// TwinCAT 3 PLC project UnitTests
// ProgramVersion: 3.1.4024.0
// libraries:
//   Tc2_Standard, * (Beckhoff Automation GmbH)
//   Tc2_System, * (Beckhoff Automation GmbH)
//   Tc2_Utilities, * (Beckhoff Automation GmbH)
//   Tc3_EventLogger, * (Beckhoff Automation GmbH)
//   Tc3_Module, * (Beckhoff Automation GmbH)
//   tcl_BaseClasses, * (Red Rock Controls Limited)
//   tcl_StringUtils, * (Red Rock Controls Limited)
//   tcl_UnitTestLibrary, * (Red Rock Controls Limited)
// project tree:
//   GVLs/ GlobalNotifications.TcGVL
//   / PlcTask.TcTTO
//   POUs/ MAIN.TcPOU
//   Unit Tests/Execution Result Aggregate/ Test_AggregateResult_Aborted.TcPOU, Test_AggregateResult_Ready.TcPOU, Test_AggregateResult_Busy.TcPOU, Test_AggregateResult_Done.TcPOU, Test_AggregateResult_Error.TcPOU, Test_AggregateResult_ErrorMsg.TcPOU, Test_AggregateResult_Starting.TcPOU, Test_AggregateResult_Aborting.TcPOU
//   Unit Tests/Execution/ Test_TExecutionWhenBusy_Abort_SelectsAborting.TcPOU, Test_TExecutionWhenBusy_SetDone_SetsDone.TcPOU, Test_TExecutionWhenReady_Start_SelectsStarting.TcPOU, Test_TExecution_SetErrorHandlesString_ErrorId.TcPOU
//   Unit Tests/Functions/ Test_ErrorIdToString.TcPOU, Test_F_DINT_TO_UDINT_Conversion.TcPOU, Test_F_Equals.TcPOU, Test_F_NotEqual.TcPOU, Test_F_UDINT_TO_DINT_Conversion.TcPOU
//   Unit Tests/Logger/ Test_TLogger_LogCritical.TcPOU, Test_TLogger_LogError.TcPOU, Test_TLogger_LogWarning.TcPOU, Test_TLogger_LogInfo.TcPOU, Test_TLogger_LogDebug.TcPOU
//   Unit Tests/Notifications/ Test_MultipleNotificationsWithStringArgs.TcPOU, Test_NotificationCountWithQueueingEnabled.TcPOU, Test_NotificationHandlerOnlyAddedOnce.TcPOU, Test_NotificationNoArgs.TcPOU, Test_NotificationWithStringArg.TcPOU
//   Unit Tests/Stream/General/ Test_TStreamBufferResizes.TcPOU
//   Unit Tests/Stream/With alignment checks/ Test_TStreamAddReadArgType_CheckAlignment.TcPOU, Test_TStreamAdd_Read_BLOB_CheckAlignment.TcPOU, Test_TStreamAdd_Read_DINT_CheckAlignment.TcPOU, Test_TStreamAdd_Read_INT_CheckAlignment.TcPOU, Test_TStreamAdd_Read_LINT_CheckAlignment.TcPOU, Test_TStreamAdd_Read_LREAL_CheckAlignment.TcPOU, Test_TStreamAdd_Read_PVOID_CheckAlignment.TcPOU, Test_TStreamAdd_Read_REAL_CheckAlignment.TcPOU, Test_TStreamAdd_Read_UDINT_CheckAlignment.TcPOU, Test_TStreamAdd_Read_UINT_CheckAlignment.TcPOU, Test_TStreamAdd_Read_ULINT_CheckAlignment.TcPOU
//   Unit Tests/Stream/With Arg Type Checking/ Test_TStreamAddReadArgType.TcPOU, Test_TStreamAdd_Read_BLOB.TcPOU, Test_TStreamAdd_Read_BOOL.TcPOU, Test_TStreamAdd_Read_BYTE.TcPOU, Test_TStreamAdd_Read_DINT.TcPOU, Test_TStreamAdd_Read_INT.TcPOU, Test_TStreamAdd_Read_LINT.TcPOU, Test_TStreamAdd_Read_LREAL.TcPOU, Test_TStreamAdd_Read_PVOID.TcPOU, Test_TStreamAdd_Read_REAL.TcPOU, Test_TStreamAdd_Read_Short_STRING.TcPOU, Test_TStreamAdd_Read_STRING.TcPOU, Test_TStreamAdd_Read_T_MaxString.TcPOU, Test_TStreamAdd_Read_UDINT.TcPOU, Test_TStreamAdd_Read_UINT.TcPOU, Test_TStreamAdd_Read_ULINT.TcPOU
//   Unit Tests/ T_TestSuite.TcPOU
// (motion and I/O tree: see PLC project tcl_baseclasses)
// real-time tasks:
//   TASK PlcTask: cycle T#10ms, priority 20, ADS port 350
//   TASK PlcTask1: cycle T#10ms, priority 21, ADS port 351

CONFIGURATION UnitTests
    RESOURCE PLC ON TwinCAT3
        TASK PlcTask(INTERVAL := T#10ms, PRIORITY := 20);
        PROGRAM PB_TestRunner WITH PlcTask : PB_TestRunner;
    END_RESOURCE
END_CONFIGURATION

// ---- GVLs/GlobalNotifications.TcGVL
{attribute 'qualified_only'}
VAR_GLOBAL
	Notification_ExecutionFailed : T_Notification;
	Notification_ExecutionAborted : T_Notification;
	
	
	
	
	
END_VAR

// ---- POUs/MAIN.TcPOU
PROGRAM MAIN
VAR
	TestSuite : T_TestSuite;
END_VAR

TestSuite.RunTests();

END_PROGRAM

// ---- Unit Tests/T_TestSuite.TcPOU
{attribute 'no_explicit_call' := 'do not call this POU directly'}
FUNCTION_BLOCK T_TestSuite
VAR
    Test_AggregateResult_Ready                      : Test_AggregateResult_Ready;
    Test_AggregateResult_Starting                   : Test_AggregateResult_Starting;
    Test_AggregateResult_Busy                       : Test_AggregateResult_Busy;
    Test_AggregateResult_Done                       : Test_AggregateResult_Done;
    Test_AggregateResult_Error                      : Test_AggregateResult_Error;
    Test_AggregateResult_ErrorMsg                   : Test_AggregateResult_ErrorMsg;
    Test_AggregateResult_Aborting                   : Test_AggregateResult_Aborting;
    Test_AggregateResult_Aborted                    : Test_AggregateResult_Aborted;
//    Test_TExecution_WhenBusy_Abort_SelectsAborting  : Test_TExecutionWhenBusy_Abort_SelectsAborting;
//    Test_TExecution_WhenBusy_SetDone_SetsDone       : Test_TExecutionWhenBusy_SetDone_SetsDone;
//    Test_TExecution_WhenReady_Start_SelectsStarting : Test_TExecutionWhenReady_Start_SelectsStarting;
//    Test_TExecution_SetErrorHandlesString_ErrorId   : Test_TExecution_SetErrorHandlesString_ErrorId;
//    Test_F_DINT_TO_UDINT_Conversion                 : Test_F_DINT_TO_UDINT_Conversion;
//    Test_F_UDINT_TO_DINT_Conversion                 : Test_F_UDINT_TO_DINT_Conversion;
//    Test_F_Equals                                   : Test_F_Equals;
//    Test_F_NotEqual                                 : Test_F_NotEqual;
//    Test_ErrorIdToString                            : Test_ErrorIdToString;
//    Test_NotificationNoArgs                         : Test_NotificationNoArgs;
//    Test_NotificationWithStringArg                  : Test_NotificationWithStringArg;
//    Test_NotificationCountWithQueueingEnabled       : Test_NotificationCountWithQueueingEnabled;
//    Test_MultipleNotificationsWithStringArgs        : Test_MultipleNotificationsWithStringArgs;
//    Test_NotificationHandlerOnlyAddedOnce           : Test_NotificationHandlerOnlyAddedOnce;

//    Test_TStreamAdd_Read_BLOB                 : Test_TStreamAdd_Read_BLOB;
//    Test_TStreamAdd_Read_BLOB_CheckAlignment  : Test_TStreamAdd_Read_BLOB_CheckAlignment;
//    Test_TStreamAdd_Read_BOOL                 : Test_TStreamAdd_Read_BOOL;
//    Test_TStreamAdd_Read_BYTE                 : Test_TStreamAdd_Read_BYTE;
//    Test_TStreamAdd_Read_DINT                 : Test_TStreamAdd_Read_DINT;
//    Test_TStreamAdd_Read_DINT_CheckAlignment  : Test_TStreamAdd_Read_DINT_CheckAlignment;
//    Test_TStreamAdd_Read_INT                  : Test_TStreamAdd_Read_INT;
//    Test_TStreamAdd_Read_INT_CheckAlignment   : Test_TStreamAdd_Read_INT_CheckAlignment;
//    Test_TStreamAdd_Read_LINT                 : Test_TStreamAdd_Read_LINT;
//    Test_TStreamAdd_Read_LINT_CheckAlignment  : Test_TStreamAdd_Read_LINT_CheckAlignment;
//    Test_TStreamAdd_Read_LREAL                : Test_TStreamAdd_Read_LREAL;
//    Test_TStreamAdd_Read_LREAL_CheckAlignment : Test_TStreamAdd_Read_LREAL_CheckAlignment;
//    Test_TStreamAdd_Read_PVOID                : Test_TStreamAdd_Read_PVOID;
//    Test_TStreamAdd_Read_PVOID_CheckAlignment : Test_TStreamAdd_Read_PVOID_CheckAlignment;
//    Test_TStreamAdd_Read_REAL                 : Test_TStreamAdd_Read_REAL;
//    Test_TStreamAdd_Read_REAL_CheckAlignment  : Test_TStreamAdd_Read_REAL_CheckAlignment;
//    Test_TStreamAdd_Read_Short_STRING         : Test_TStreamAdd_Read_Short_STRING;
//    Test_TStreamAdd_Read_STRING               : Test_TStreamAdd_Read_STRING;
//    Test_TStreamAdd_Read_T_MaxString          : Test_TStreamAdd_Read_T_MaxString;
//    Test_TStreamAdd_Read_UDINT                : Test_TStreamAdd_Read_UDINT;
//    Test_TStreamAdd_Read_UDINT_CheckAlignment : Test_TStreamAdd_Read_UDINT_CheckAlignment;
//    Test_TStreamAdd_Read_UINT                 : Test_TStreamAdd_Read_UINT;
//    Test_TStreamAdd_Read_UINT_CheckAlignment  : Test_TStreamAdd_Read_UINT_CheckAlignment;
//    Test_TStreamAdd_Read_ULINT                : Test_TStreamAdd_Read_ULINT;
//    Test_TStreamAdd_Read_ULINT_CheckAlignment : Test_TStreamAdd_Read_ULINT_CheckAlignment;
//    Test_TStreamAddReadArgType                : Test_TStreamAddReadArgType;
//    Test_TStreamAddReadArgType_CheckAlignment : Test_TStreamAddReadArgType_CheckAlignment;
//    Test_TStreamBufferResizes                 : Test_TStreamBufferResizes;

//    Test_TLogger_LogCritical : Test_TLogger_LogCritical;
//    Test_TLogger_LogError    : Test_TLogger_LogError;
//    Test_TLogger_LogWarning  : Test_TLogger_LogWarning;
//    Test_TLogger_LogInfo     : Test_TLogger_LogInfo;
//    Test_TLogger_LogDebug    : Test_TLogger_LogDebug;
END_VAR

METHOD RunTests
VAR_INPUT
END_VAR
Test_AggregateResult_Ready                     		.RunTest();
Test_AggregateResult_Starting                       .RunTest();
Test_AggregateResult_Busy                           .RunTest();
Test_AggregateResult_Done                           .RunTest();
Test_AggregateResult_Error                          .RunTest();
Test_AggregateResult_ErrorMsg                       .RunTest();
Test_AggregateResult_Aborting                       .RunTest();
Test_AggregateResult_Aborted                        .RunTest();
//Test_TExecution_WhenBusy_Abort_SelectsAborting      .RunTest();
//Test_TExecution_WhenBusy_SetDone_SetsDone           .RunTest();
//Test_TExecution_WhenReady_Start_SelectsStarting     .RunTest();
//Test_TExecution_SetErrorHandlesString_ErrorId       .RunTest();
//Test_F_DINT_TO_UDINT_Conversion                     .RunTest();
//Test_F_UDINT_TO_DINT_Conversion                     .RunTest();
//Test_F_Equals                                       .RunTest();
//Test_F_NotEqual                                     .RunTest();
//Test_ErrorIdToString                                .RunTest();
//Test_NotificationNoArgs                             .RunTest();
//Test_NotificationWithStringArg                      .RunTest();
//Test_NotificationCountWithQueueingEnabled           .RunTest();
//Test_MultipleNotificationsWithStringArgs            .RunTest();
//Test_NotificationHandlerOnlyAddedOnce               .RunTest();

//Test_TStreamAdd_Read_BLOB                			.RunTest();
//Test_TStreamAdd_Read_BLOB_CheckAlignment            .RunTest();
//Test_TStreamAdd_Read_BOOL                           .RunTest();
//Test_TStreamAdd_Read_BYTE                           .RunTest();
//Test_TStreamAdd_Read_DINT                           .RunTest();
//Test_TStreamAdd_Read_DINT_CheckAlignment            .RunTest();
//Test_TStreamAdd_Read_INT                            .RunTest();
//Test_TStreamAdd_Read_INT_CheckAlignment             .RunTest();
//Test_TStreamAdd_Read_LINT                           .RunTest();
//Test_TStreamAdd_Read_LINT_CheckAlignment            .RunTest();
//Test_TStreamAdd_Read_LREAL                          .RunTest();
//Test_TStreamAdd_Read_LREAL_CheckAlignment           .RunTest();
//Test_TStreamAdd_Read_PVOID                          .RunTest();
//Test_TStreamAdd_Read_PVOID_CheckAlignment           .RunTest();
//Test_TStreamAdd_Read_REAL                           .RunTest();
//Test_TStreamAdd_Read_REAL_CheckAlignment            .RunTest();
//Test_TStreamAdd_Read_Short_STRING                   .RunTest();
//Test_TStreamAdd_Read_STRING                         .RunTest();
//Test_TStreamAdd_Read_T_MaxString                    .RunTest();
//Test_TStreamAdd_Read_UDINT                          .RunTest();
//Test_TStreamAdd_Read_UDINT_CheckAlignment           .RunTest();
//Test_TStreamAdd_Read_UINT                           .RunTest();
//Test_TStreamAdd_Read_UINT_CheckAlignment            .RunTest();
//Test_TStreamAdd_Read_ULINT                          .RunTest();
//Test_TStreamAdd_Read_ULINT_CheckAlignment           .RunTest();
//Test_TStreamAddReadArgType                          .RunTest();
//Test_TStreamAddReadArgType_CheckAlignment           .RunTest();
//Test_TStreamBufferResizes                           .RunTest();

//Test_TLogger_LogCritical .RunTest();
//Test_TLogger_LogError    .RunTest();
//Test_TLogger_LogWarning  .RunTest();
//Test_TLogger_LogInfo     .RunTest();
//Test_TLogger_LogDebug    .RunTest();
END_METHOD

END_FUNCTION_BLOCK

// ---- Unit Tests/Execution Result Aggregate/Test_AggregateResult_Ready.TcPOU
FUNCTION_BLOCK Test_AggregateResult_Ready EXTENDS T_UnitTestBase
VAR
    ResultAggregate : T_ResultAggregate;
    Execution1      : T_Execution;
    Execution2      : T_Execution;
    Execution3      : T_Execution;
END_VAR

{attribute 'analysis' := '-33'} // inhibit unused variable warning
METHOD RunTest
IF Retest THEN
    SUPER^.Init();
END_IF

IF TestCompleted THEN
    RETURN;
END_IF

F_Inc(CycleCount);
IF CycleCount > 1000 THEN
    Fail(Message := 'Timeout');
END_IF

ResultAggregate.Clear();

ResultAggregate.AddResult(Execution1);
ResultAggregate.AddResult(Execution2);
ResultAggregate.AddResult(Execution3);

AssertIsTrue(Condition := ResultAggregate.Ready = TRUE,
             Message   := 'ResultAggregate.Ready is not true');

Execution1.Start();
Execution1.SetBusy();

AssertIsTrue(Condition := ResultAggregate.Ready = FALSE,
             Message   := 'ResultAggregate.Ready is not false');

TestCompleted := TRUE;
END_METHOD

END_FUNCTION_BLOCK

// ---- Unit Tests/Execution Result Aggregate/Test_AggregateResult_Starting.TcPOU
FUNCTION_BLOCK Test_AggregateResult_Starting EXTENDS T_UnitTestBase
VAR
    ResultAggregate : T_ResultAggregate;
    Execution1      : T_Execution;
    Execution2      : T_Execution;
    Execution3      : T_Execution;
END_VAR

{attribute 'analysis' := '-33'} // inhibit unused variable warning
METHOD RunTest
IF Retest THEN
    SUPER^.Init();
END_IF

IF TestCompleted THEN
    RETURN;
END_IF

F_Inc(CycleCount);
IF CycleCount > 1000 THEN
    Fail(Message := 'Timeout');
END_IF

ResultAggregate.Clear();

ResultAggregate.AddResult(Execution1);
ResultAggregate.AddResult(Execution2);
ResultAggregate.AddResult(Execution3);

AssertIsTrue(Condition := ResultAggregate.Starting = FALSE,
             Message   := 'ResultAggregate.Starting is not false');

Execution1.Start();

AssertIsTrue(Condition := ResultAggregate.Starting = TRUE,
             Message   := 'ResultAggregate.Starting is false');

TestCompleted := TRUE;
END_METHOD

END_FUNCTION_BLOCK

// ---- Unit Tests/Execution Result Aggregate/Test_AggregateResult_Busy.TcPOU
FUNCTION_BLOCK Test_AggregateResult_Busy EXTENDS T_UnitTestBase
VAR
	ResultAggregate : T_ResultAggregate;
	Execution1 : T_Execution;
	Execution2 : T_Execution;
	Execution3 : T_Execution;
END_VAR

{attribute 'analysis' := '-33'} // inhibit unused variable warning
METHOD RunTest
IF Retest THEN
    SUPER^.Init();
END_IF

IF TestCompleted THEN
    RETURN;
END_IF

F_Inc(CycleCount);
IF CycleCount > 1000 THEN
    Fail(Message := 'Timeout');
END_IF

ResultAggregate.Clear();

ResultAggregate.AddResult(Execution1);
ResultAggregate.AddResult(Execution2);
ResultAggregate.AddResult(Execution3);

AssertIsTrue(Condition := ResultAggregate.Busy = FALSE,
             Message   := 'ResultAggregate.Busy is not false');

Execution1.Start();
Execution1.SetBusy();

AssertIsTrue(Condition := ResultAggregate.Busy = TRUE,
             Message   := 'ResultAggregate.Busy is false');

TestCompleted := TRUE;
END_METHOD

END_FUNCTION_BLOCK

// ---- Unit Tests/Execution Result Aggregate/Test_AggregateResult_Done.TcPOU
FUNCTION_BLOCK Test_AggregateResult_Done EXTENDS T_UnitTestBase
VAR
	ResultAggregate : T_ResultAggregate;
	Execution1 : T_Execution;
	Execution2 : T_Execution;
	Execution3 : T_Execution;
END_VAR

{attribute 'analysis' := '-33'} // inhibit unused variable warning
METHOD RunTest
IF Retest THEN
    SUPER^.Init();
END_IF

IF TestCompleted THEN
    RETURN;
END_IF

F_Inc(CycleCount);
IF CycleCount > 1000 THEN
    Fail(Message := 'Timeout');
END_IF

ResultAggregate.Clear();

ResultAggregate.AddResult(Execution1);
ResultAggregate.AddResult(Execution2);
ResultAggregate.AddResult(Execution3);

Execution1.Start();
Execution1.SetBusy();
Execution1.SetDone();

Execution2.Start();
Execution2.SetBusy();
Execution2.SetDone();

AssertIsTrue(Condition := ResultAggregate.Done = FALSE,
             Message   := 'ResultAggregate.Done is not false');

Execution3.Start();
Execution3.SetBusy();
Execution3.SetDone();

AssertIsTrue(Condition := ResultAggregate.Done = TRUE,
             Message   := 'ResultAggregate.Done is false');

TestCompleted := TRUE;
END_METHOD

END_FUNCTION_BLOCK

// ---- Unit Tests/Execution Result Aggregate/Test_AggregateResult_Error.TcPOU
FUNCTION_BLOCK Test_AggregateResult_Error EXTENDS T_UnitTestBase
VAR
	ResultAggregate : T_ResultAggregate;
	Execution1 : T_Execution;
	Execution2 : T_Execution;
	Execution3 : T_Execution;
END_VAR

{attribute 'analysis' := '-33'} // inhibit unused variable warning
METHOD RunTest
IF Retest THEN
    SUPER^.Init();
END_IF

IF TestCompleted THEN
    RETURN;
END_IF

F_Inc(CycleCount);
IF CycleCount > 1000 THEN
    Fail(Message := 'Timeout');
END_IF

ResultAggregate.Clear();

ResultAggregate.AddResult(Execution1);
ResultAggregate.AddResult(Execution2);
ResultAggregate.AddResult(Execution3);

Execution1.Start();
Execution1.SetBusy();

AssertIsTrue(Condition := ResultAggregate.Error = FALSE,
             Message   := 'ResultAggregate.Error is not false');

Execution3.Start();
Execution3.SetBusy();
Execution3.SetError('Expected Error Message');

AssertIsTrue(Condition := ResultAggregate.Error = TRUE,
             Message   := 'ResultAggregate.Error is false');

TestCompleted := TRUE;
END_METHOD

END_FUNCTION_BLOCK

// ---- Unit Tests/Execution Result Aggregate/Test_AggregateResult_ErrorMsg.TcPOU
FUNCTION_BLOCK Test_AggregateResult_ErrorMsg EXTENDS T_UnitTestBase
VAR
	ResultAggregate : T_ResultAggregate;
	Execution1 : T_Execution;
	Execution2 : T_Execution;
	Execution3 : T_Execution;
END_VAR

{attribute 'analysis' := '-33'} // inhibit unused variable warning
METHOD RunTest
IF Retest THEN
    SUPER^.Init();
END_IF

IF TestCompleted THEN
    RETURN;
END_IF

F_Inc(CycleCount);
IF CycleCount > 1000 THEN
    Fail(Message := 'Timeout');
END_IF

ResultAggregate.Clear();

ResultAggregate.AddResult(Execution1);
ResultAggregate.AddResult(Execution2);
ResultAggregate.AddResult(Execution3);

Execution1.Start();
Execution1.SetBusy();
Execution1.SetDone();

Execution2.Start();
Execution2.SetBusy();
Execution2.SetDone();

AssertIsTrue(Condition := ResultAggregate.ErrorMsg = '',
             Message   := 'ResultAggregate.ErrorMsg is not blank');

Execution3.Start();
Execution3.SetBusy();
Execution3.SetError('Expected Error Message');

AssertIsTrue(Condition := ResultAggregate.ErrorMsg = 'Expected Error Message',
             Message   := 'ResultAggregate.ErrorMsg is incorrect');

TestCompleted := TRUE;
END_METHOD

END_FUNCTION_BLOCK

// ---- Unit Tests/Execution Result Aggregate/Test_AggregateResult_Aborting.TcPOU
FUNCTION_BLOCK Test_AggregateResult_Aborting EXTENDS T_UnitTestBase
VAR
    ResultAggregate : T_ResultAggregate;
    Execution1      : T_Execution;
    Execution2      : T_Execution;
    Execution3      : T_Execution;
END_VAR

{attribute 'analysis' := '-33'} // inhibit unused variable warning
METHOD RunTest
IF Retest THEN
    SUPER^.Init();
END_IF

IF TestCompleted THEN
    RETURN;
END_IF

F_Inc(CycleCount);
IF CycleCount > 1000 THEN
    Fail(Message := 'Timeout');
END_IF

ResultAggregate.Clear();

ResultAggregate.AddResult(Execution1);
ResultAggregate.AddResult(Execution2);
ResultAggregate.AddResult(Execution3);

AssertIsTrue(Condition := ResultAggregate.Aborting = FALSE,
             Message   := 'ResultAggregate.Aborting is not false');

Execution3.Start();
Execution3.SetBusy();
Execution3.Abort();

AssertIsTrue(Condition := ResultAggregate.Aborting = TRUE,
             Message   := 'ResultAggregate.Aborting is false');

TestCompleted := TRUE;
END_METHOD

END_FUNCTION_BLOCK

// ---- Unit Tests/Execution Result Aggregate/Test_AggregateResult_Aborted.TcPOU
FUNCTION_BLOCK Test_AggregateResult_Aborted EXTENDS T_UnitTestBase
VAR
    ResultAggregate : T_ResultAggregate;
    Execution1      : T_Execution;
    Execution2      : T_Execution;
    Execution3      : T_Execution;
END_VAR

{attribute 'analysis' := '-33'} // inhibit unused variable warning
METHOD RunTest
IF Retest THEN
    SUPER^.Init();
END_IF

IF TestCompleted THEN
    RETURN;
END_IF

F_Inc(CycleCount);
IF CycleCount > 1000 THEN
    Fail(Message := 'Timeout');
END_IF

ResultAggregate.Clear();

ResultAggregate.AddResult(Execution1);
ResultAggregate.AddResult(Execution2);
ResultAggregate.AddResult(Execution3);

AssertIsTrue(Condition := ResultAggregate.Aborted = FALSE,
             Message   := 'ResultAggregate.Aborted is not false');

Execution1.Start();
Execution1.SetBusy();
Execution1.Abort();
Execution1.SetAborted();

Execution2.Start();
Execution2.SetBusy();
Execution2.Abort();
Execution2.SetAborted();

Execution3.Start();
Execution3.SetBusy();
Execution3.Abort();
Execution3.SetAborted();

AssertIsTrue(Condition := ResultAggregate.Aborted,
             Message   := 'ResultAggregate.Aborting is false');

TestCompleted := TRUE;
END_METHOD

END_FUNCTION_BLOCK

// ---- Unit Tests/Execution/Test_TExecutionWhenBusy_Abort_SelectsAborting.TcPOU
FUNCTION_BLOCK Test_TExecutionWhenBusy_Abort_SelectsAborting EXTENDS T_UnitTestbase
VAR
    Execution : T_Execution;
END_VAR

{attribute 'analysis' := '-33'} // inhibit unused variable warning
METHOD RunTest
IF Retest THEN
    SUPER^.Init();
END_IF

IF TestCompleted THEN
    RETURN;
END_IF

F_Inc(CycleCount);
IF CycleCount > 1000 THEN
    Fail(Message := 'Timeout');
END_IF

Execution.Start();
Execution.SetBusy();
Execution.Abort();

AssertIsTrue(Condition := Execution.Aborting,
             Message   := 'Execution.Aborting not true');

TestCompleted := TRUE;
END_METHOD

END_FUNCTION_BLOCK

// ---- Unit Tests/Execution/Test_TExecutionWhenBusy_SetDone_SetsDone.TcPOU
FUNCTION_BLOCK Test_TExecutionWhenBusy_SetDone_SetsDone EXTENDS T_UnitTestbase
VAR
    Execution : T_Execution;
END_VAR

{attribute 'analysis' := '-33'} // inhibit unused variable warning
METHOD RunTest
IF Retest THEN
    SUPER^.Init();
END_IF

IF TestCompleted THEN
    RETURN;
END_IF

F_Inc(CycleCount);
IF CycleCount > 1000 THEN
    Fail(Message := 'Timeout');
END_IF

// Test...
Execution.Start();
Execution.SetBusy();
Execution.SetDone();

AssertIsTrue(Condition := Execution.Done,
             Message   := 'Execution.Done not true');

AssertIsTrue(Condition := Execution.Ready,
             Message   := 'Execution.Ready not true');

TestCompleted := TRUE;
END_METHOD

END_FUNCTION_BLOCK

// ---- Unit Tests/Execution/Test_TExecutionWhenReady_Start_SelectsStarting.TcPOU
FUNCTION_BLOCK Test_TExecutionWhenReady_Start_SelectsStarting EXTENDS T_UnitTestbase
VAR
    Execution : T_Execution;
END_VAR

{attribute 'analysis' := '-33'} // inhibit unused variable warning
METHOD RunTest
IF Retest THEN
    SUPER^.Init();
END_IF

IF TestCompleted THEN
    RETURN;
END_IF

F_Inc(CycleCount);
IF CycleCount > 1000 THEN
    Fail(Message := 'Timeout');
END_IF

// Test...
Execution.Start();

AssertIsTrue(Condition := Execution.Starting,
             Message   := 'Execution.Starting not true');

TestCompleted := TRUE;
END_METHOD

END_FUNCTION_BLOCK

// ---- Unit Tests/Execution/Test_TExecution_SetErrorHandlesString_ErrorId.TcPOU
FUNCTION_BLOCK Test_TExecution_SetErrorHandlesString_ErrorId EXTENDS T_UnitTestBase
VAR
    Execution : T_Execution;
END_VAR
VAR
    ErrorId : STRING := 'Custom error message';
END_VAR

{attribute 'analysis' := '-33'} // inhibit unused variable warning
METHOD RunTest
VAR
    ErrorMsg : STRING := 'Expected error message';
END_VAR
IF Retest THEN
    SUPER^.Init();
END_IF

IF TestCompleted THEN
    RETURN;
END_IF

F_Inc(CycleCount);
IF CycleCount > 1000 THEN
    Fail(Message := 'Timeout');
END_IF

Execution.Start();
Execution.SetBusy();
Execution.SetError(ErrorMsg);

AssertIsTrue(Condition := Execution.ErrorMsg = 'Expected error message',
             Message   := 'Execution.ErrorMsg not correct');

TestCompleted := TRUE;
END_METHOD

END_FUNCTION_BLOCK

// ---- Unit Tests/Functions/Test_ErrorIdToString.TcPOU
FUNCTION_BLOCK Test_ErrorIdToString EXTENDS T_UnitTestBase
VAR_INPUT
END_VAR
VAR_OUTPUT
END_VAR
VAR
END_VAR

{attribute 'analysis' := '-33'} // inhibit unused variable warning
METHOD RunTest
IF Retest THEN
    SUPER^.Init();
END_IF

IF TestCompleted THEN
    RETURN;
END_IF

F_Inc(CycleCount);
IF CycleCount > 1000 THEN
    Fail(Message := 'Timeout');
END_IF

AssertEquals_STRING(Expected := 'Error 0x12BD',
                      Actual   := F_ErrorIdToString(16#12BD),
                      Message  := 'F_ErrorIdToString(16#12BD)');

AssertEquals_STRING(Expected := 'Error 0x12345678',
                      Actual   := F_ErrorIdToString(16#12345678),
                      Message  := 'F_ErrorIdToString(16#12345678)');

AssertEquals_STRING(Expected := 'Error 0x00FF',
                      Actual   := F_ErrorIdToString(16#FF),
                      Message  := 'F_ErrorIdToString(16#FF)');

AssertEquals_STRING(Expected := 'Error 0x0011 - No debugging available',
                      Actual   := F_ErrorIdToString(16#11),
                      Message  := 'F_ErrorIdToString(16#11)');

TestCompleted := TRUE;
END_METHOD

END_FUNCTION_BLOCK

// ---- Unit Tests/Functions/Test_F_DINT_TO_UDINT_Conversion.TcPOU
FUNCTION_BLOCK Test_F_DINT_TO_UDINT_Conversion EXTENDS T_UnitTestBase
VAR
    InputValue     : DINT;
    ConvertedValue : UDINT;
END_VAR

{attribute 'analysis' := '-33'} // inhibit unused variable warning
METHOD RunTest
IF Retest THEN
    SUPER^.Init();
END_IF

IF TestCompleted THEN
    RETURN;
END_IF

F_Inc(CycleCount);
IF CycleCount > 1000 THEN
    Fail(Message := 'Timeout');
END_IF

InputValue     := 2147483648;                  // too big
ConvertedValue := F_UDINT_TO_DINT(InputValue); // limit to largest DINT

AssertEquals_DINT(Expected := 2147483647,
                  Actual   := ConvertedValue,
                  Message  := 'ConvertedValue is not correct');

TestCompleted := TRUE;
END_METHOD

END_FUNCTION_BLOCK

// ---- Unit Tests/Functions/Test_F_Equals.TcPOU
FUNCTION_BLOCK Test_F_Equals EXTENDS T_UnitTestBase
VAR
	
END_VAR

{attribute 'analysis' := '-33'} // inhibit unused variable warning
METHOD RunTest
IF Retest THEN
    SUPER^.Init();
END_IF

IF TestCompleted THEN
    RETURN;
END_IF

F_Inc(CycleCount);
IF CycleCount > 1000 THEN
    Fail(Message := 'Timeout');
END_IF

AssertIsTrue(Condition := F_Equals(1.000_005,
                                   1.000_004,
                                   0.000_002),
             Message := 'F_Equals does not return TRUE');

AssertIsTrue(Condition := NOT F_Equals(1.000_005,
                                   1.000_003,
                                   0.000_001),
             Message := 'F_Equals does not return FALSE');

TestCompleted := TRUE;
END_METHOD

END_FUNCTION_BLOCK

// ---- Unit Tests/Functions/Test_F_NotEqual.TcPOU
FUNCTION_BLOCK Test_F_NotEqual EXTENDS T_UnitTestBase
VAR

END_VAR

{attribute 'analysis' := '-33'} // inhibit unused variable warning
METHOD RunTest
IF Retest THEN
    SUPER^.Init();
END_IF

IF TestCompleted THEN
    RETURN;
END_IF

F_Inc(CycleCount);
IF CycleCount > 1000 THEN
    Fail(Message := 'Timeout');
END_IF

AssertIsTrue(Condition := F_NotEqual(1.000_005,
                                     1.000_003,
                                     0.000_001),
             Message := 'F_NotEquals returns incorrect result');

AssertIsTrue(Condition := NOT F_NotEqual(1.000_005,
                                         1.000_004,
                                         0.000_002),
             Message := 'F_NotEquals returns incorrect result');

TestCompleted := TRUE;
END_METHOD

END_FUNCTION_BLOCK

// ---- Unit Tests/Functions/Test_F_UDINT_TO_DINT_Conversion.TcPOU
FUNCTION_BLOCK Test_F_UDINT_TO_DINT_Conversion EXTENDS T_UnitTestBase
VAR
    InputValue     : UDINT;
    ConvertedValue : DINT;
END_VAR

{attribute 'analysis' := '-33'} // inhibit unused variable warning
METHOD RunTest
IF Retest THEN
    SUPER^.Init();
END_IF

IF TestCompleted THEN
    RETURN;
END_IF

F_Inc(CycleCount);
IF CycleCount > 1000 THEN
    Fail(Message := 'Timeout');
END_IF

InputValue     := UDINT#2147483648;            // too big
ConvertedValue := F_UDINT_TO_DINT(InputValue); // limit to largest DINT

AssertIsTrue(Condition := (ConvertedValue = 2147483647),
             Message   := 'F_UDINT_TO_DINT returns incorrect value');

TestCompleted := TRUE;
END_METHOD

END_FUNCTION_BLOCK

// ---- Unit Tests/Logger/Test_TLogger_LogCritical.TcPOU
FUNCTION_BLOCK Test_TLogger_LogCritical EXTENDS T_UnitTestBase
VAR
    SourceInfo : FB_TcSourceInfo;
END_VAR

{attribute 'analysis' := '-33'} // inhibit unused variable warning
METHOD RunTest
VAR
    ErrorMsg : STRING := 'Expected error message';
END_VAR
IF Retest THEN
    SUPER^.Init();
END_IF

IF TestCompleted THEN
    RETURN;
END_IF

F_Inc(CycleCount);
IF CycleCount > 1000 THEN
    Fail(Message := 'Timeout');
END_IF

SourceInfo.sName := 'ExpectedSourceName';
DefaultLogger.LogCritical(SourceInfo,'Expected critical message1');
DefaultLogger.LogCritical(SourceInfo,'Expected critical message2');

TestCompleted := TRUE;
END_METHOD

END_FUNCTION_BLOCK

// ---- Unit Tests/Logger/Test_TLogger_LogError.TcPOU
FUNCTION_BLOCK Test_TLogger_LogError EXTENDS T_UnitTestBase
VAR
    SourceInfo : FB_TcSourceInfo;
END_VAR

{attribute 'analysis' := '-33'} // inhibit unused variable warning
METHOD RunTest
VAR
    ErrorMsg : STRING := 'Expected error message';
END_VAR
IF Retest THEN
    SUPER^.Init();
END_IF

IF TestCompleted THEN
    RETURN;
END_IF

F_Inc(CycleCount);
IF CycleCount > 1000 THEN
    Fail(Message := 'Timeout');
END_IF

SourceInfo.sName := 'ExpectedSourceName';
DefaultLogger.LogError(SourceInfo,'Expected error message1');
DefaultLogger.LogError(SourceInfo,'Expected error message2');

TestCompleted := TRUE;
END_METHOD

END_FUNCTION_BLOCK

// ---- Unit Tests/Logger/Test_TLogger_LogWarning.TcPOU
FUNCTION_BLOCK Test_TLogger_LogWarning EXTENDS T_UnitTestBase
VAR
    SourceInfo : FB_TcSourceInfo;
END_VAR

{attribute 'analysis' := '-33'} // inhibit unused variable warning
METHOD RunTest
VAR
    ErrorMsg : STRING := 'Expected error message';
END_VAR
IF Retest THEN
    SUPER^.Init();
END_IF

IF TestCompleted THEN
    RETURN;
END_IF

F_Inc(CycleCount);
IF CycleCount > 1000 THEN
    Fail(Message := 'Timeout');
END_IF

SourceInfo.sName := 'ExpectedSourceName';
DefaultLogger.LogWarning(SourceInfo,'Expected warning error message1');
DefaultLogger.LogWarning(SourceInfo,'Expected warning error message2');

TestCompleted := TRUE;
END_METHOD

END_FUNCTION_BLOCK

// ---- Unit Tests/Logger/Test_TLogger_LogInfo.TcPOU
FUNCTION_BLOCK Test_TLogger_LogInfo EXTENDS T_UnitTestBase
VAR
    SourceInfo : FB_TcSourceInfo;
END_VAR

{attribute 'analysis' := '-33'} // inhibit unused variable warning
METHOD RunTest
VAR
    ErrorMsg : STRING := 'Expected error message';
END_VAR
IF Retest THEN
    SUPER^.Init();
END_IF

IF TestCompleted THEN
    RETURN;
END_IF

F_Inc(CycleCount);
IF CycleCount > 1000 THEN
    Fail(Message := 'Timeout');
END_IF

SourceInfo.sName := 'ExpectedSourceName';
DefaultLogger.LogInfo(SourceInfo,'Expected info message1');
DefaultLogger.LogInfo(SourceInfo,'Expected info message2');

TestCompleted := TRUE;
END_METHOD

END_FUNCTION_BLOCK

// ---- Unit Tests/Logger/Test_TLogger_LogDebug.TcPOU
FUNCTION_BLOCK Test_TLogger_LogDebug EXTENDS T_UnitTestBase
VAR
    SourceInfo : FB_TcSourceInfo;
END_VAR

{attribute 'analysis' := '-33'} // inhibit unused variable warning
METHOD RunTest
VAR
    ErrorMsg : STRING := 'Expected error message';
END_VAR
IF Retest THEN
    SUPER^.Init();
END_IF

IF TestCompleted THEN
    RETURN;
END_IF

F_Inc(CycleCount);
IF CycleCount > 1000 THEN
    Fail(Message := 'Timeout');
END_IF

SourceInfo.sName := 'ExpectedSourceName';
DefaultLogger.LogDebug(SourceInfo,'Expected debug message1');
DefaultLogger.LogDebug(SourceInfo,'Expected debug message2');

TestCompleted := TRUE;
END_METHOD

END_FUNCTION_BLOCK

// ---- Unit Tests/Notifications/Test_MultipleNotificationsWithStringArgs.TcPOU
{attribute 'hide'}
FUNCTION_BLOCK Test_MultipleNotificationsWithStringArgs EXTENDS T_UnitTestBase
VAR
    Notification        : T_Notification;
    NotificationHandler : T_NotificationHandler;

    IsRaised          : BOOL;
    NotificationCount : DINT;
END_VAR

{attribute 'analysis' := '-33'} // inhibit unused variable warning
METHOD RunTest
IF Retest THEN
    SUPER^.Init();
END_IF

IF TestCompleted THEN
    RETURN;
END_IF

F_Inc(CycleCount);
IF CycleCount > 1000 THEN
    Fail(Message := 'Timeout');
END_IF

NotificationHandler.NotificationQueueingEnabled := TRUE; // Notification Queuing requires care to ensure all notifications are handled, so disabled by default!

IsRaised          := FALSE;
NotificationCount := 0;

Notification.ClearNotificationHandlers().AddNotificationHandler(NotificationHandler);
Notification.Args.Init(8);

Notification.Args.Clear()
    .Add_INT(1234).Add_STRING('String1');

Notification.Raise();

Notification.Args.Clear()
    .Add_INT(5678).Add_STRING('String2');

Notification.Raise();

AssertEquals_DINT(Expected := 2,
                  Actual   := NotificationHandler.NotificationCount,
                  Message  := 'Handler.NotificationCount is not 2');

AssertIsTrue(Condition := NotificationHandler.IsRaised(),
             Message   := 'NotificationHandler.IsRaised() returns false');

AssertEquals_DINT(Expected := 1,
                  Actual   := NotificationHandler.NotificationCount,
                  Message  := 'Handler.NotificationCount is not 1');

AssertEquals_DINT(Expected := 1234,
                  Actual   := NotificationHandler.Args.Read_INT(),
                  Message  := 'Handler.Args.Read_INT() is not 1234');

AssertEquals_STRING(Expected := 'String1',
                    Actual   := NotificationHandler.Args.Read_STRING(),
                    Message  := 'Handler.Args.Read_STRING() returns incorrect value');

AssertIsTrue(Condition := NotificationHandler.IsRaised(),
             Message   := 'Handler.IsRaised() returns false');

AssertEquals_DINT(Expected := 0,
                  Actual   := NotificationHandler.NotificationCount,
                  Message  := 'Handler.NotificationCount is not 0');

AssertEquals_DINT(Expected := 5678,
                  Actual   := NotificationHandler.Args.Read_INT(),
                  Message  := 'Handler.Args.Read_INT() does not return 5678');

AssertEquals_STRING(Expected := 'String2',
                    Actual   := NotificationHandler.Args.Read_STRING(),
                    Message  := 'Handler.Args.Read_STRING() does not return String2');

AssertIsTrue(Condition := NotificationHandler.IsRaised() = FALSE,
             Message   := 'Handler.IsRaised() return true');

TestCompleted := TRUE;
END_METHOD

END_FUNCTION_BLOCK

// ---- Unit Tests/Notifications/Test_NotificationCountWithQueueingEnabled.TcPOU
FUNCTION_BLOCK Test_NotificationCountWithQueueingEnabled EXTENDS T_UnitTestBase
VAR
    Notification   : T_Notification;
    NotificationHandler : T_NotificationHandler;
    IsRaised : BOOL;
END_VAR

{attribute 'analysis' := '-33'} // inhibit unused variable warning
METHOD RunTest
IF Retest THEN
    SUPER^.Init();
END_IF

IF TestCompleted THEN
    RETURN;
END_IF

F_Inc(CycleCount);
IF CycleCount > 1000 THEN
    Fail(Message := 'Timeout');
END_IF

NotificationHandler.NotificationQueueingEnabled := TRUE; // Notification Queuing requires care to ensure all notifications are handled, so disabled by default!

Notification.ClearNotificationHandlers().AddNotificationHandler(NotificationHandler);

Notification.Raise();
Notification.Raise();
Notification.Raise();

AssertEquals_DINT(Expected := 3,
                  Actual   := NotificationHandler.NotificationCount,
                  Message  := 'Handler.NotificationCount is not 3');

AssertIsTrue(Condition := NotificationHandler.IsRaised(),
             Message   := 'IsRaised() does not return true');

AssertEquals_DINT(Expected := 2,
                  Actual   := NotificationHandler.NotificationCount,
                  Message  := 'Handler.NotificationCount is not 2');

AssertIsTrue(Condition := NotificationHandler.IsRaised(),
             Message   := 'IsRaised() does not return true');

AssertEquals_DINT(Expected := 1,
                  Actual   := NotificationHandler.NotificationCount,
                  Message  := 'Handler.NotificationCount is not 1');

IsRaised := NotificationHandler.IsRaised();

AssertIsTrue(Condition := IsRaised,
             Message   := 'IsRaised is false');

AssertEquals_DINT(Expected     := 0,
                  Actual       := NotificationHandler.NotificationCount,
                  Message := 'Handler.NotificationCount is not 0');

AssertIsTrue(Condition    := NotificationHandler.IsRaised() = FALSE,
             Message := 'Handler.IsRaised() is not false');

TestCompleted := TRUE;
END_METHOD

END_FUNCTION_BLOCK

// ---- Unit Tests/Notifications/Test_NotificationHandlerOnlyAddedOnce.TcPOU
FUNCTION_BLOCK Test_NotificationHandlerOnlyAddedOnce EXTENDS T_UnitTestBase
VAR
    Notification        : T_Notification;
    NotificationHandler : T_NotificationHandler;
    IsRaised            : BOOL;
END_VAR

{attribute 'analysis' := '-33'} // inhibit unused variable warning
METHOD RunTest
IF Retest THEN
    SUPER^.Init();
END_IF

IF TestCompleted THEN
    RETURN;
END_IF

F_Inc(CycleCount);
IF CycleCount > 1000 THEN
    Fail(Message := 'Timeout');
END_IF

Notification
    .ClearNotificationHandlers()
    .AddNotificationHandler(NotificationHandler)
    .AddNotificationHandler(NotificationHandler);

Notification.Raise();
IsRaised := NotificationHandler.IsRaised();

AssertIsTrue(Condition := IsRaised = TRUE,
             Message   := 'IsRaised is not true');

IsRaised := NotificationHandler.IsRaised();

AssertIsTrue(Condition := IsRaised = FALSE,
             Message   := 'IsRaised is not false');

TestCompleted := TRUE;
END_METHOD

END_FUNCTION_BLOCK

// ---- Unit Tests/Notifications/Test_NotificationNoArgs.TcPOU
FUNCTION_BLOCK Test_NotificationNoArgs EXTENDS T_UnitTestBase
VAR
    Notification        : T_Notification;
    NotificationHandler : T_NotificationHandler;
    IsRaised            : BOOL;
END_VAR

{attribute 'analysis' := '-33'} // inhibit unused variable warning
METHOD RunTest
IF Retest THEN
    SUPER^.Init();
END_IF

IF TestCompleted THEN
    RETURN;
END_IF

F_Inc(CycleCount);
IF CycleCount > 1000 THEN
    Fail(Message := 'Timeout');
END_IF

Notification.ClearNotificationHandlers().AddNotificationHandler(NotificationHandler);

Notification.Raise();
IsRaised := NotificationHandler.IsRaised();

AssertIsTrue(Condition := IsRaised,
             Message   := 'IsRaised is not true');

TestCompleted := TRUE;
END_METHOD

END_FUNCTION_BLOCK

// ---- Unit Tests/Notifications/Test_NotificationWithStringArg.TcPOU
{attribute 'hide'}
FUNCTION_BLOCK Test_NotificationWithStringArg EXTENDS T_UnitTestBase
VAR
    Notification        : T_Notification;
    NotificationHandler : T_NotificationHandler;

    ResultString : T_MaxString;
    Args         : I_StreamReader;
    IsRaised     : BOOL;
END_VAR

{attribute 'analysis' := '-33'} // inhibit unused variable warning
METHOD RunTest
IF Retest THEN
    SUPER^.Init();
END_IF

IF TestCompleted THEN
    RETURN;
END_IF

F_Inc(CycleCount);
IF CycleCount > 1000 THEN
    Fail(Message := 'Timeout');
END_IF

Notification.ClearNotificationHandlers().AddNotificationHandler(NotificationHandler);
Notification.Args.Init(81);

Notification.Args.Clear().Add_STRING('Big long string passed to the notification handler for later use');
Notification.Raise();

IF NotificationHandler.IsRaised() THEN
    Args         := NotificationHandler.Args;
    ResultString := Args.Read_STRING();
END_IF

AssertEquals_STRING(Expected := 'Big long string passed to the notification handler for later use',
                    Actual   := ResultString,
                    Message  := 'ResultString is not correct');

TestCompleted := TRUE;
END_METHOD

END_FUNCTION_BLOCK

// ---- Unit Tests/Stream/General/Test_TStreamBufferResizes.TcPOU
FUNCTION_BLOCK Test_TStreamBufferResizes EXTENDS T_UnitTestBase
VAR
    Stream : T_Stream(StreamLength := 2);
END_VAR

{attribute 'analysis' := '-33'} // inhibit unused variable warning
METHOD RunTest
IF Retest THEN
    SUPER^.Init();
END_IF

IF TestCompleted THEN
    RETURN;
END_IF

F_Inc(CycleCount);
IF CycleCount > 1000 THEN
    Fail(Message := 'Timeout');
END_IF

Stream.Init(2);

Stream.Add_INT(1234);
Stream.Add_INT(1235);
Stream.Add_INT(1236);
Stream.Add_INT(1237);

AssertEquals_UDINT(Expected     := 8,
                   Actual       := Stream.WritePosition,
                   Message := 'Stream.WritePosition');

AssertEquals_UDINT(Expected     := 8,
                   Actual       := Stream.StreamLength,
                   Message := 'Stream.StreamLength');

Stream.SetReadPosition(0);

AssertEquals_INT(Expected     := 1234,
                 Actual       := Stream.Read_INT(),
                 Message := 'Stream.ReadInt()');

AssertEquals_UDINT(Expected     := 2,
                   Actual       := Stream.ReadPosition,
                   Message := 'Stream.ReadPosition');

TestCompleted := TRUE;
END_METHOD

END_FUNCTION_BLOCK

// ---- Unit Tests/Stream/With alignment checks/Test_TStreamAddReadArgType_CheckAlignment.TcPOU
FUNCTION_BLOCK Test_TStreamAddReadArgType_CheckAlignment EXTENDS T_UnitTestBase
VAR
    Stream : T_Stream(StreamLength := 2);
END_VAR

{attribute 'analysis' := '-33'} // inhibit unused variable warning
METHOD RunTest
IF Retest THEN
    SUPER^.Init();
END_IF

IF TestCompleted THEN
    RETURN;
END_IF

F_Inc(CycleCount);
IF CycleCount > 1000 THEN
    Fail(Message := 'Timeout');
END_IF

Stream.Init(2);

Stream.Add_BYTE(123); // add a byte to test alignment checks...
Stream.SetNextArgTypeId(E_ArgTypeId.Type_LINT);

AssertEquals_UDINT(Expected := 4,
                   Actual   := Stream.WritePosition,
                   Message  := 'Stream.WritePosition');

Stream.SetReadPosition(0);

Stream.Read_BYTE();

AssertEquals_INT(Expected := E_ArgTypeId.Type_LINT,
                 Actual   := Stream.GetNextArgTypeId(),
                 Message  := 'Stream.GetNextArgTypeId()');

AssertEquals_UDINT(Expected := 4,
                   Actual   := Stream.ReadPosition,
                   Message  := 'Stream.ReadPosition');

TestCompleted := TRUE;
END_METHOD

END_FUNCTION_BLOCK

// ---- Unit Tests/Stream/With alignment checks/Test_TStreamAdd_Read_BLOB_CheckAlignment.TcPOU
FUNCTION_BLOCK Test_TStreamAdd_Read_BLOB_CheckAlignment EXTENDS T_UnitTestBase
VAR
    Stream : T_Stream(StreamLength := 2);
    Now    : TIMESTRUCT := (wDay := 23,
        wMonth := 12,
        wYear := 1945,
        wHour := 22,
        wMinute := 20,
        wSecond := 18);
    NowFromStream : TIMESTRUCT;

    LREAL_Value : LREAL := 1.234;
END_VAR

{attribute 'analysis' := '-33'} // inhibit unused variable warning
METHOD RunTest
IF Retest THEN
    SUPER^.Init();
END_IF

IF TestCompleted THEN
    RETURN;
END_IF

F_Inc(CycleCount);
IF CycleCount > 1000 THEN
    Fail(Message := 'Timeout');
END_IF

Stream.Init(2);
NowFromStream.wDay    := 0;
NowFromStream.wMonth  := 0;
NowFromStream.wYear   := 0;
NowFromStream.wHour   := 0;
NowFromStream.wMinute := 0;
NowFromStream.wSecond := 0;

Stream.Add_BYTE(123);// add a byte to test alignment checks...
Stream.Add_BLOB(Now);

Stream.SetReadPosition(0);
Stream.Read_BYTE();
Stream.Read_BLOB(NowFromStream);

// check the value...
AssertEquals_ANY(Expected     := Now,
                            Actual       := NowFromStream,
                            Message := 'NowFromStream');

// check we are at the end of the stream..							
AssertEquals_UDINT(Expected     := Stream.StreamLength,
                             Actual       := Stream.ReadPosition,
                             Message := 'Stream.ReadPosition');

TestCompleted := TRUE;
END_METHOD

END_FUNCTION_BLOCK

// ---- Unit Tests/Stream/With alignment checks/Test_TStreamAdd_Read_DINT_CheckAlignment.TcPOU
FUNCTION_BLOCK Test_TStreamAdd_Read_DINT_CheckAlignment EXTENDS T_UnitTestBase
VAR
    Stream  : T_Stream(StreamLength := 2);
    ArgType : E_ArgTypeId := E_ArgTypeId.Type_DINT;
END_VAR

{attribute 'analysis' := '-33'} // inhibit unused variable warning
METHOD RunTest
IF Retest THEN
    SUPER^.Init();
END_IF

IF TestCompleted THEN
    RETURN;
END_IF

F_Inc(CycleCount);
IF CycleCount > 1000 THEN
    Fail(Message := 'Timeout');
END_IF

Stream.Init(2);

Stream.Add_BYTE(123);// add a byte to test alignment checks...
Stream.Add_DINT(12345678);

Stream.SetReadPosition(0);

Stream.Read_BYTE();

// check next value...	
AssertEquals_DINT(Expected     := 12345678,
                            Actual       := Stream.Read_DINT(),
                            Message := 'Stream.Read_DINT()');

// check we are at the end of the stream..							
AssertEquals_UDINT(Expected     := Stream.StreamLength,
                             Actual       := Stream.ReadPosition,
                             Message := 'Stream.ReadPosition');

TestCompleted := TRUE;
END_METHOD

END_FUNCTION_BLOCK

// ---- Unit Tests/Stream/With alignment checks/Test_TStreamAdd_Read_INT_CheckAlignment.TcPOU
FUNCTION_BLOCK Test_TStreamAdd_Read_INT_CheckAlignment EXTENDS T_UnitTestBase
VAR
    Stream  : T_Stream(StreamLength := 2);
    ArgType : E_ArgTypeId := E_ArgTypeId.Type_INT;
END_VAR

{attribute 'analysis' := '-33'} // inhibit unused variable warning
METHOD RunTest
IF Retest THEN
    SUPER^.Init();
END_IF

IF TestCompleted THEN
    RETURN;
END_IF

F_Inc(CycleCount);
IF CycleCount > 1000 THEN
    Fail(Message := 'Timeout');
END_IF

Stream.Init(2);

Stream.Add_BYTE(123);// add a byte to test alignment checks...
Stream.Add_INT(1234);

Stream.SetReadPosition(0);

Stream.Read_BYTE();

// check next value...	
AssertEquals_INT(Expected     := 1234,
                           Actual       := Stream.Read_INT(),
                           Message := 'Stream.Read_INT()');

// check we are at the end of the stream..							
AssertEquals_UDINT(Expected     := Stream.StreamLength,
                             Actual       := Stream.ReadPosition,
                             Message := 'Stream.ReadPosition');

TestCompleted := TRUE;
END_METHOD

END_FUNCTION_BLOCK

// ---- Unit Tests/Stream/With alignment checks/Test_TStreamAdd_Read_LINT_CheckAlignment.TcPOU
FUNCTION_BLOCK Test_TStreamAdd_Read_LINT_CheckAlignment EXTENDS T_UnitTestBase
VAR
    Stream  : T_Stream(StreamLength := 2);
    ArgType : E_ArgTypeId := E_ArgTypeId.Type_LINT;
END_VAR

{attribute 'analysis' := '-33'} // inhibit unused variable warning
METHOD RunTest
IF Retest THEN
    SUPER^.Init();
END_IF

IF TestCompleted THEN
    RETURN;
END_IF

F_Inc(CycleCount);
IF CycleCount > 1000 THEN
    Fail(Message := 'Timeout');
END_IF

Stream.Init(2);

Stream.Add_BYTE(123);// add a byte to test alignment checks...
Stream.Add_LINT(123456789);

Stream.SetReadPosition(0);

Stream.Read_BYTE();

// check next value...	
AssertEquals_LINT(Expected     := 123456789,
                            Actual       := Stream.Read_LINT(),
                            Message := 'Stream.Read_LINT()');

// check we are at the end of the stream..							
AssertEquals_UDINT(Expected     := Stream.StreamLength,
                             Actual       := Stream.ReadPosition,
                             Message := 'Stream.ReadPosition');

TestCompleted := TRUE;
END_METHOD

END_FUNCTION_BLOCK

// ---- Unit Tests/Stream/With alignment checks/Test_TStreamAdd_Read_LREAL_CheckAlignment.TcPOU
FUNCTION_BLOCK Test_TStreamAdd_Read_LREAL_CheckAlignment EXTENDS T_UnitTestBase
VAR
    Stream  : T_Stream(StreamLength := 2);
    ArgType : E_ArgTypeId := E_ArgTypeId.Type_LREAL;
END_VAR

{attribute 'analysis' := '-33'} // inhibit unused variable warning
METHOD RunTest
IF Retest THEN
    SUPER^.Init();
END_IF

IF TestCompleted THEN
    RETURN;
END_IF

F_Inc(CycleCount);
IF CycleCount > 1000 THEN
    Fail(Message := 'Timeout');
END_IF

Stream.Init(2);

Stream.Add_BYTE(123);// add a byte to test alignment checks...
Stream.Add_LREAL(1.234567891234);

Stream.SetReadPosition(0);

Stream.Read_BYTE();

// check next value...	
AssertEquals_LREAL(Expected     := 1.234567891234,
                             Actual       := Stream.Read_LREAL(),
                             Delta        := 0.000000000001,
                             Message := 'Stream.Read_LREAL()');

// check we are at the end of the stream..							
AssertEquals_UDINT(Expected     := Stream.StreamLength,
                             Actual       := Stream.ReadPosition,
                             Message := 'Stream.ReadPosition');

TestCompleted := TRUE;
END_METHOD

END_FUNCTION_BLOCK

// ---- Unit Tests/Stream/With alignment checks/Test_TStreamAdd_Read_PVOID_CheckAlignment.TcPOU
FUNCTION_BLOCK Test_TStreamAdd_Read_PVOID_CheckAlignment EXTENDS T_UnitTestBase
VAR
    Stream  : T_Stream(StreamLength := 2);
    ArgType : E_ArgTypeId := E_ArgTypeId.Type_PVOID;
    Bob     : INT;
END_VAR

{attribute 'analysis' := '-33'} // inhibit unused variable warning
METHOD RunTest
IF Retest THEN
    SUPER^.Init();
END_IF

IF TestCompleted THEN
    RETURN;
END_IF

F_Inc(CycleCount);
IF CycleCount > 1000 THEN
    Fail(Message := 'Timeout');
END_IF

Stream.Init(2);

Stream.Add_BYTE(123);// add a byte to test alignment checks...
Stream.Add_PVOID(ADR(Bob));

Stream.SetReadPosition(0);

Stream.Read_BYTE();

// check next value...	
AssertEquals_PVOID(Expected     := ADR(Bob),
                             Actual       := Stream.Read_PVOID(),
                             Message := 'Stream.Read_PVOID()');

// check we are at the end of the stream..							
AssertEquals_UDINT(Expected     := Stream.StreamLength,
                             Actual       := Stream.ReadPosition,
                             Message := 'Stream.ReadPosition');

TestCompleted := TRUE;
END_METHOD

END_FUNCTION_BLOCK

// ---- Unit Tests/Stream/With alignment checks/Test_TStreamAdd_Read_REAL_CheckAlignment.TcPOU
FUNCTION_BLOCK Test_TStreamAdd_Read_REAL_CheckAlignment EXTENDS T_UnitTestBase
VAR
    Stream  : T_Stream(StreamLength := 2);
    ArgType : E_ArgTypeId := E_ArgTypeId.Type_REAL;
END_VAR

{attribute 'analysis' := '-33'} // inhibit unused variable warning
METHOD RunTest
IF Retest THEN
    SUPER^.Init();
END_IF

IF TestCompleted THEN
    RETURN;
END_IF

F_Inc(CycleCount);
IF CycleCount > 1000 THEN
    Fail(Message := 'Timeout');
END_IF

Stream.Init(2);

Stream.Add_BYTE(123);// add a byte to test alignment checks...
Stream.Add_REAL(1.234567);

Stream.SetReadPosition(0);

Stream.Read_BYTE();

// check next value...	
AssertEquals_REAL(Expected     := 1.234567,
                            Actual       := Stream.Read_REAL(),
                            Delta        := 0.000001,
                            Message := 'Stream.Read_REAL()');

// check we are at the end of the stream..							
AssertEquals_UDINT(Expected     := Stream.StreamLength,
                             Actual       := Stream.ReadPosition,
                             Message := 'Stream.ReadPosition');

TestCompleted := TRUE;
END_METHOD

END_FUNCTION_BLOCK

// ---- Unit Tests/Stream/With alignment checks/Test_TStreamAdd_Read_UDINT_CheckAlignment.TcPOU
FUNCTION_BLOCK Test_TStreamAdd_Read_UDINT_CheckAlignment EXTENDS T_UnitTestBase
VAR
    Stream  : T_Stream(StreamLength := 2);
    ArgType : E_ArgTypeId := E_ArgTypeId.Type_UDINT;
END_VAR

{attribute 'analysis' := '-33'} // inhibit unused variable warning
METHOD RunTest
IF Retest THEN
    SUPER^.Init();
END_IF

IF TestCompleted THEN
    RETURN;
END_IF

F_Inc(CycleCount);
IF CycleCount > 1000 THEN
    Fail(Message := 'Timeout');
END_IF

Stream.Init(2);

Stream.Add_BYTE(123);// add a byte to test alignment checks...
Stream.Add_UDINT(12345678);

Stream.SetReadPosition(0);

Stream.Read_BYTE();

// check next value...	
AssertEquals_UDINT(Expected     := 12345678,
                             Actual       := Stream.Read_UDINT(),
                             Message := 'Stream.Read_UDINT()');

// check we are at the end of the stream..							
AssertEquals_UDINT(Expected     := Stream.StreamLength,
                             Actual       := Stream.ReadPosition,
                             Message := 'Stream.ReadPosition');

TestCompleted := TRUE;
END_METHOD

END_FUNCTION_BLOCK

// ---- Unit Tests/Stream/With alignment checks/Test_TStreamAdd_Read_UINT_CheckAlignment.TcPOU
FUNCTION_BLOCK Test_TStreamAdd_Read_UINT_CheckAlignment EXTENDS T_UnitTestBase
VAR
    Stream  : T_Stream(StreamLength := 2);
    ArgType : E_ArgTypeId := E_ArgTypeId.Type_UINT;
END_VAR

{attribute 'analysis' := '-33'} // inhibit unused variable warning
METHOD RunTest
IF Retest THEN
    SUPER^.Init();
END_IF

IF TestCompleted THEN
    RETURN;
END_IF

F_Inc(CycleCount);
IF CycleCount > 1000 THEN
    Fail(Message := 'Timeout');
END_IF

Stream.Init(2);

Stream.Add_BYTE(123);// add a byte to test alignment checks...
Stream.Add_UINT(4567);

Stream.SetReadPosition(0);

Stream.Read_BYTE();

// check next value...	
AssertEquals_UINT(Expected     := 4567,
                            Actual       := Stream.Read_UINT(),
                            Message := 'Stream.Read_UINT()');

// check we are at the end of the stream..							
AssertEquals_UDINT(Expected     := Stream.StreamLength,
                             Actual       := Stream.ReadPosition,
                             Message := 'Stream.ReadPosition');

TestCompleted := TRUE;
END_METHOD

END_FUNCTION_BLOCK

// ---- Unit Tests/Stream/With alignment checks/Test_TStreamAdd_Read_ULINT_CheckAlignment.TcPOU
FUNCTION_BLOCK Test_TStreamAdd_Read_ULINT_CheckAlignment EXTENDS T_UnitTestBase
VAR
    Stream  : T_Stream(StreamLength := 2);
    ArgType : E_ArgTypeId := E_ArgTypeId.Type_ULINT;
END_VAR

{attribute 'analysis' := '-33'} // inhibit unused variable warning
METHOD RunTest
IF Retest THEN
    SUPER^.Init();
END_IF

IF TestCompleted THEN
    RETURN;
END_IF

F_Inc(CycleCount);
IF CycleCount > 1000 THEN
    Fail(Message := 'Timeout');
END_IF


Stream.Init(2);

Stream.Add_BYTE(123); // add a byte to test alignment checks...
Stream.Add_ULINT(123456789);

Stream.SetReadPosition(0);

Stream.Read_BYTE();

// check next value...	
AssertEquals_ULINT(Expected     := 123456789,
                   Actual       := Stream.Read_ULINT(),
                   Message := 'Stream.Read_ULINT()');

// check we are at the end of the stream..							
AssertEquals_UDINT(Expected     := Stream.StreamLength,
                   Actual       := Stream.ReadPosition,
                   Message := 'Stream.ReadPosition');

TestCompleted := TRUE;
END_METHOD

END_FUNCTION_BLOCK

// ---- Unit Tests/Stream/With Arg Type Checking/Test_TStreamAddReadArgType.TcPOU
FUNCTION_BLOCK Test_TStreamAddReadArgType EXTENDS T_UnitTestBase
VAR
    Stream : T_Stream(StreamLength := 2);
END_VAR

{attribute 'analysis' := '-33'} // inhibit unused variable warning
METHOD RunTest
IF Retest THEN
    SUPER^.Init();
END_IF

IF TestCompleted THEN
    RETURN;
END_IF

F_Inc(CycleCount);
IF CycleCount > 1000 THEN
    Fail(Message := 'Timeout');
END_IF

Stream.Init(2);

Stream.SetNextArgTypeId(E_ArgTypeId.Type_LINT);

AssertEquals_UDINT(Expected     := 2,
                             Actual       := Stream.WritePosition,
                             Message := 'Stream.WritePosition');

Stream.SetReadPosition(0);

AssertEquals_INT(Expected     := E_ArgTypeId.Type_LINT,
                           Actual       := Stream.GetNextArgTypeId(),
                           Message := 'Stream.GetNextArgTypeId()');

AssertEquals_UDINT(Expected     := 2,
                             Actual       := Stream.ReadPosition,
                             Message := 'Stream.ReadPosition');

TestCompleted := TRUE;
END_METHOD

END_FUNCTION_BLOCK

// ---- Unit Tests/Stream/With Arg Type Checking/Test_TStreamAdd_Read_BLOB.TcPOU
FUNCTION_BLOCK Test_TStreamAdd_Read_BLOB EXTENDS T_UnitTestBase
VAR
    Stream : T_Stream(StreamLength := 2);
    Now    : TIMESTRUCT := (wDay := 23,
        wMonth := 12,
        wYear := 1945,
        wHour := 22,
        wMinute := 20,
        wSecond := 18);
    NowFromStream : TIMESTRUCT;

    LREAL_Value : LREAL := 1.234;
END_VAR

{attribute 'analysis' := '-33'} // inhibit unused variable warning
METHOD RunTest
IF Retest THEN
    SUPER^.Init();
END_IF

IF TestCompleted THEN
    RETURN;
END_IF

F_Inc(CycleCount);
IF CycleCount > 1000 THEN
    Fail(Message := 'Timeout');
END_IF

Stream.Init(2);
NowFromStream.wDay    := 0;
NowFromStream.wMonth  := 0;
NowFromStream.wYear   := 0;
NowFromStream.wHour   := 0;
NowFromStream.wMinute := 0;
NowFromStream.wSecond := 0;

Stream.SetNextArgTypeId(E_ArgTypeId.Type_Blob);
Stream.Add_BLOB(Now);

Stream.SetReadPosition(0);

IF Stream.GetNextArgTypeId() = E_ArgTypeId.Type_Blob THEN
    Stream.Read_BLOB(NowFromStream);
END_IF

// check the value...
AssertEquals_ANY(Expected     := Now,
                            Actual       := NowFromStream,
                            Message := 'NowFromStream');

// check we are at the end of the stream..							
AssertEquals_UDINT(Expected     := Stream.StreamLength,
                             Actual       := Stream.ReadPosition,
                             Message := 'Stream.ReadPosition');

TestCompleted := TRUE;
END_METHOD

END_FUNCTION_BLOCK

// ---- Unit Tests/Stream/With Arg Type Checking/Test_TStreamAdd_Read_BOOL.TcPOU
FUNCTION_BLOCK Test_TStreamAdd_Read_BOOL EXTENDS T_UnitTestBase
VAR
    Stream  : T_Stream(StreamLength := 2);
    ArgType : E_ArgTypeId := E_ArgTypeId.Type_BOOL;
END_VAR

{attribute 'analysis' := '-33'} // inhibit unused variable warning
METHOD RunTest
IF Retest THEN
    SUPER^.Init();
END_IF

IF TestCompleted THEN
    RETURN;
END_IF

F_Inc(CycleCount);
IF CycleCount > 1000 THEN
    Fail(Message := 'Timeout');
END_IF

Stream.Init(2);

// add a bool...
Stream.SetNextArgTypeId(ArgType);
Stream.Add_BOOL(TRUE);

Stream.SetReadPosition(0);

// check next arg type is correct...
AssertEquals_INT(Expected     := ArgType,
                           Actual       := Stream.GetNextArgTypeId(),
                           Message := 'Stream.GetNextArgTypeId()');

// check next value...	
AssertEquals_BOOL(Expected     := TRUE,
                            Actual       := Stream.Read_BOOL(),
                            Message := 'Stream.Read_BOOL()');

// check we are at the end of the stream..							
AssertEquals_UDINT(Expected     := Stream.StreamLength,
                             Actual       := Stream.ReadPosition,
                             Message := 'Stream.ReadPosition');

TestCompleted := TRUE;
END_METHOD

END_FUNCTION_BLOCK

// ---- Unit Tests/Stream/With Arg Type Checking/Test_TStreamAdd_Read_BYTE.TcPOU
FUNCTION_BLOCK Test_TStreamAdd_Read_BYTE EXTENDS T_UnitTestBase
VAR
    Stream  : T_Stream(StreamLength := 2);
    ArgType : E_ArgTypeId := E_ArgTypeId.Type_BYTE;
END_VAR

{attribute 'analysis' := '-33'} // inhibit unused variable warning
METHOD RunTest
IF Retest THEN
    SUPER^.Init();
END_IF

IF TestCompleted THEN
    RETURN;
END_IF

F_Inc(CycleCount);
IF CycleCount > 1000 THEN
    Fail(Message := 'Timeout');
END_IF

Stream.Init(2);

// add a byte...
Stream.SetNextArgTypeId(ArgType);
Stream.Add_BYTE(123);

Stream.SetReadPosition(0);

// check next arg type is correct...
AssertEquals_INT(Expected     := ArgType,
                           Actual       := Stream.GetNextArgTypeId(),
                           Message := 'Stream.GetNextArgTypeId()');

// check next value...	
AssertEquals_BYTE(Expected     := 123,
                            Actual       := Stream.Read_BYTE(),
                            Message := 'Stream.Read_BYTE()');

// check we are at the end of the stream..							
AssertEquals_UDINT(Expected     := Stream.StreamLength,
                             Actual       := Stream.ReadPosition,
                             Message := 'Stream.ReadPosition');

TestCompleted := TRUE;
END_METHOD

END_FUNCTION_BLOCK

// ---- Unit Tests/Stream/With Arg Type Checking/Test_TStreamAdd_Read_DINT.TcPOU
FUNCTION_BLOCK Test_TStreamAdd_Read_DINT EXTENDS T_UnitTestBase
VAR
    Stream  : T_Stream(StreamLength := 2);
    ArgType : E_ArgTypeId := E_ArgTypeId.Type_DINT;
END_VAR

{attribute 'analysis' := '-33'} // inhibit unused variable warning
METHOD RunTest
IF Retest THEN
    SUPER^.Init();
END_IF

IF TestCompleted THEN
    RETURN;
END_IF

F_Inc(CycleCount);
IF CycleCount > 1000 THEN
    Fail(Message := 'Timeout');
END_IF

Stream.Init(2);

// add a DINT...
Stream.SetNextArgTypeId(ArgType);
Stream.Add_DINT(12345678);

Stream.SetReadPosition(0);

// check next arg type is correct...
AssertEquals_INT(Expected     := ArgType,
                           Actual       := Stream.GetNextArgTypeId(),
                           Message := 'Stream.GetNextArgTypeId()');

// check next value...	
AssertEquals_DINT(Expected     := 12345678,
                            Actual       := Stream.Read_DINT(),
                            Message := 'Stream.Read_DINT()');

// check we are at the end of the stream..							
AssertEquals_UDINT(Expected     := Stream.StreamLength,
                             Actual       := Stream.ReadPosition,
                             Message := 'Stream.ReadPosition');

TestCompleted := TRUE;
END_METHOD

END_FUNCTION_BLOCK

// ---- Unit Tests/Stream/With Arg Type Checking/Test_TStreamAdd_Read_INT.TcPOU
FUNCTION_BLOCK Test_TStreamAdd_Read_INT EXTENDS T_UnitTestBase
VAR
    Stream  : T_Stream(StreamLength := 2);
    ArgType : E_ArgTypeId := E_ArgTypeId.Type_INT;
END_VAR

{attribute 'analysis' := '-33'} // inhibit unused variable warning
METHOD RunTest
IF Retest THEN
    SUPER^.Init();
END_IF

IF TestCompleted THEN
    RETURN;
END_IF

F_Inc(CycleCount);
IF CycleCount > 1000 THEN
    Fail(Message := 'Timeout');
END_IF

Stream.Init(2);

// add an INT...
Stream.SetNextArgTypeId(ArgType);
Stream.Add_INT(1234);

Stream.SetReadPosition(0);

// check next arg type is correct...
AssertEquals_INT(Expected     := ArgType,
                           Actual       := Stream.GetNextArgTypeId(),
                           Message := 'Stream.GetNextArgTypeId()');

// check next value...	
AssertEquals_INT(Expected     := 1234,
                           Actual       := Stream.Read_INT(),
                           Message := 'Stream.Read_INT()');

// check we are at the end of the stream..							
AssertEquals_UDINT(Expected     := Stream.StreamLength,
                             Actual       := Stream.ReadPosition,
                             Message := 'Stream.ReadPosition');

TestCompleted := TRUE;
END_METHOD

END_FUNCTION_BLOCK

// ---- Unit Tests/Stream/With Arg Type Checking/Test_TStreamAdd_Read_LINT.TcPOU
FUNCTION_BLOCK Test_TStreamAdd_Read_LINT EXTENDS T_UnitTestBase
VAR
    Stream  : T_Stream(StreamLength := 2);
    ArgType : E_ArgTypeId := E_ArgTypeId.Type_LINT;
END_VAR

{attribute 'analysis' := '-33'} // inhibit unused variable warning
METHOD RunTest
IF Retest THEN
    SUPER^.Init();
END_IF

IF TestCompleted THEN
    RETURN;
END_IF

F_Inc(CycleCount);
IF CycleCount > 1000 THEN
    Fail(Message := 'Timeout');
END_IF

Stream.Init(2);

// add a LINT...
Stream.SetNextArgTypeId(ArgType);
Stream.Add_LINT(123456789);

Stream.SetReadPosition(0);

// check next arg type is correct...
AssertEquals_INT(Expected     := ArgType,
                           Actual       := Stream.GetNextArgTypeId(),
                           Message := 'Stream.GetNextArgTypeId()');

// check next value...	
AssertEquals_LINT(Expected     := 123456789,
                            Actual       := Stream.Read_LINT(),
                            Message := 'Stream.Read_LINT()');

// check we are at the end of the stream..							
AssertEquals_UDINT(Expected     := Stream.StreamLength,
                             Actual       := Stream.ReadPosition,
                             Message := 'Stream.ReadPosition');

TestCompleted := TRUE;
END_METHOD

END_FUNCTION_BLOCK

// ---- Unit Tests/Stream/With Arg Type Checking/Test_TStreamAdd_Read_LREAL.TcPOU
FUNCTION_BLOCK Test_TStreamAdd_Read_LREAL EXTENDS T_UnitTestBase
VAR
    Stream  : T_Stream(StreamLength := 2);
    ArgType : E_ArgTypeId := E_ArgTypeId.Type_LREAL;
END_VAR

{attribute 'analysis' := '-33'} // inhibit unused variable warning
METHOD RunTest
IF Retest THEN
    SUPER^.Init();
END_IF

IF TestCompleted THEN
    RETURN;
END_IF

F_Inc(CycleCount);
IF CycleCount > 1000 THEN
    Fail(Message := 'Timeout');
END_IF

Stream.Init(2);

// add a LREAL...
Stream.SetNextArgTypeId(ArgType);
Stream.Add_LREAL(1.234567891234);

Stream.SetReadPosition(0);

// check next arg type is correct...
AssertEquals_INT(Expected     := ArgType,
                           Actual       := Stream.GetNextArgTypeId(),
                           Message := 'Stream.GetNextArgTypeId()');

// check next value...	
AssertEquals_LREAL(Expected     := 1.234567891234,
                             Actual       := Stream.Read_LREAL(),
                             Delta        := 0.000000000001,
                             Message := 'Stream.Read_LREAL()');

// check we are at the end of the stream..							
AssertEquals_UDINT(Expected     := Stream.StreamLength,
                             Actual       := Stream.ReadPosition,
                             Message := 'Stream.ReadPosition');

TestCompleted := TRUE;
END_METHOD

END_FUNCTION_BLOCK

// ---- Unit Tests/Stream/With Arg Type Checking/Test_TStreamAdd_Read_PVOID.TcPOU
FUNCTION_BLOCK Test_TStreamAdd_Read_PVOID EXTENDS T_UnitTestBase
VAR
    Stream  : T_Stream(StreamLength := 2);
    ArgType : E_ArgTypeId := E_ArgTypeId.Type_PVOID;
    Bob     : INT;
END_VAR

{attribute 'analysis' := '-33'} // inhibit unused variable warning
METHOD RunTest
IF Retest THEN
    SUPER^.Init();
END_IF

IF TestCompleted THEN
    RETURN;
END_IF

F_Inc(CycleCount);
IF CycleCount > 1000 THEN
    Fail(Message := 'Timeout');
END_IF

Stream.Init(2);

// add a pointer...
Stream.SetNextArgTypeId(ArgType);
Stream.Add_PVOID(ADR(Bob));

Stream.SetReadPosition(0);

// check next arg type is correct...
AssertEquals_INT(Expected     := ArgType,
                           Actual       := Stream.GetNextArgTypeId(),
                           Message := 'Stream.GetNextArgTypeId()');

// check next value...	
AssertEquals_PVOID(Expected     := ADR(Bob),
                             Actual       := Stream.Read_PVOID(),
                             Message := 'Stream.Read_PVOID()');

// check we are at the end of the stream..							
AssertEquals_UDINT(Expected     := Stream.StreamLength,
                             Actual       := Stream.ReadPosition,
                             Message := 'Stream.ReadPosition');

TestCompleted := TRUE;
END_METHOD

END_FUNCTION_BLOCK

// ---- Unit Tests/Stream/With Arg Type Checking/Test_TStreamAdd_Read_REAL.TcPOU
FUNCTION_BLOCK Test_TStreamAdd_Read_REAL EXTENDS T_UnitTestBase
VAR
    Stream  : T_Stream(StreamLength := 2);
    ArgType : E_ArgTypeId := E_ArgTypeId.Type_REAL;
END_VAR

{attribute 'analysis' := '-33'} // inhibit unused variable warning
METHOD RunTest
IF Retest THEN
    SUPER^.Init();
END_IF

IF TestCompleted THEN
    RETURN;
END_IF

F_Inc(CycleCount);
IF CycleCount > 1000 THEN
    Fail(Message := 'Timeout');
END_IF

Stream.Init(2);

// add a REAL...
Stream.SetNextArgTypeId(ArgType);
Stream.Add_REAL(1.234567);

Stream.SetReadPosition(0);

// check next arg type is correct...
AssertEquals_INT(Expected     := ArgType,
                           Actual       := Stream.GetNextArgTypeId(),
                           Message := 'Stream.GetNextArgTypeId()');

// check next value...	
AssertEquals_REAL(Expected     := 1.234567,
                            Actual       := Stream.Read_REAL(),
                            Delta        := 0.000001,
                            Message := 'Stream.Read_REAL()');

// check we are at the end of the stream..							
AssertEquals_UDINT(Expected     := Stream.StreamLength,
                             Actual       := Stream.ReadPosition,
                             Message := 'Stream.ReadPosition');

TestCompleted := TRUE;
END_METHOD

END_FUNCTION_BLOCK

// ---- Unit Tests/Stream/With Arg Type Checking/Test_TStreamAdd_Read_Short_STRING.TcPOU
FUNCTION_BLOCK Test_TStreamAdd_Read_Short_STRING EXTENDS T_UnitTestBase
VAR
    Stream     : T_Stream(StreamLength := 2);
    ArgType    : E_ArgTypeId := E_ArgTypeId.Type_STRING;
    TestString : STRING(10)  := '0123456789';
END_VAR

{attribute 'analysis' := '-33'} // inhibit unused variable warning
METHOD RunTest
IF Retest THEN
    SUPER^.Init();
END_IF

IF TestCompleted THEN
    RETURN;
END_IF

F_Inc(CycleCount);
IF CycleCount > 1000 THEN
    Fail(Message := 'Timeout');
END_IF


Stream.Init(2);

// add a STRING...
Stream.SetNextArgTypeId(ArgType);
Stream.Add_STRING(TestString);

Stream.SetReadPosition(0);

// check next arg type is correct...
AssertEquals_INT(Expected     := ArgType,
                           Actual       := Stream.GetNextArgTypeId(),
                           Message := 'Stream.GetNextArgTypeId()');

// check next value...	
AssertEquals_STRING(Expected     := TestString,
                              Actual       := Stream.Read_STRING(),
                              Message := 'Stream.Read_STRING()');

// check we are at the end of the stream..							
AssertEquals_UDINT(Expected     := Stream.StreamLength,
                             Actual       := Stream.ReadPosition,
                             Message := 'Stream.ReadPosition');

TestCompleted := TRUE;
END_METHOD

END_FUNCTION_BLOCK

// ---- Unit Tests/Stream/With Arg Type Checking/Test_TStreamAdd_Read_STRING.TcPOU
FUNCTION_BLOCK Test_TStreamAdd_Read_STRING EXTENDS T_UnitTestBase
VAR
    Stream     : T_Stream(StreamLength := 2);
    ArgType    : E_ArgTypeId := E_ArgTypeId.Type_STRING;
    TestString : STRING      := '111111111 222222222 333333333 444444444 555555555 666666666 777777777 888888888 ';
END_VAR

{attribute 'analysis' := '-33'} // inhibit unused variable warning
METHOD RunTest
IF Retest THEN
    SUPER^.Init();
END_IF

IF TestCompleted THEN
    RETURN;
END_IF

F_Inc(CycleCount);
IF CycleCount > 1000 THEN
    Fail(Message := 'Timeout');
END_IF

Stream.Init(2);

// add a STRING...
Stream.SetNextArgTypeId(ArgType);
Stream.Add_STRING(TestString);

Stream.SetReadPosition(0);

// check next arg type is correct...
AssertEquals_INT(Expected     := ArgType,
                           Actual       := Stream.GetNextArgTypeId(),
                           Message := 'Stream.GetNextArgTypeId()');

// check next value...	
AssertEquals_STRING(Expected     := TestString,
                              Actual       := Stream.Read_STRING(),
                              Message := 'Stream.Read_STRING()');

// check we are at the end of the stream..							
AssertEquals_UDINT(Expected     := Stream.StreamLength,
                             Actual       := Stream.ReadPosition,
                             Message := 'Stream.ReadPosition');

TestCompleted := TRUE;
END_METHOD

END_FUNCTION_BLOCK

// ---- Unit Tests/Stream/With Arg Type Checking/Test_TStreamAdd_Read_T_MaxString.TcPOU
FUNCTION_BLOCK Test_TStreamAdd_Read_T_MaxString EXTENDS T_UnitTestBase
VAR
    Stream     : T_Stream(StreamLength := 2);
    ArgType    : E_ArgTypeId := E_ArgTypeId.Type_STRING;
    TestString : T_MaxString := '111111111 222222222 333333333 444444444 555555555 666666666 777777777 888888888 999999999 ';
END_VAR

{attribute 'analysis' := '-33'} // inhibit unused variable warning
METHOD RunTest
IF Retest THEN
    SUPER^.Init();
END_IF

IF TestCompleted THEN
    RETURN;
END_IF

F_Inc(CycleCount);
IF CycleCount > 1000 THEN
    Fail(Message := 'Timeout');
END_IF

Stream.Init(2);

// add a STRING...
Stream.SetNextArgTypeId(ArgType);
Stream.Add_String(TestString);

Stream.SetReadPosition(0);

// check next arg type is correct...
AssertEquals_INT(Expected     := ArgType,
                           Actual       := Stream.GetNextArgTypeId(),
                           Message := 'Stream.GetNextArgTypeId()');

// check next value...	
AssertEquals_STRING(Expected     := TestString,
                              Actual       := Stream.Read_String(),
                              Message := 'Stream.Read_String()');

// check we are at the end of the stream..							
AssertEquals_UDINT(Expected     := Stream.StreamLength,
                             Actual       := Stream.ReadPosition,
                             Message := 'Stream.ReadPosition');

TestCompleted := TRUE;
END_METHOD

END_FUNCTION_BLOCK

// ---- Unit Tests/Stream/With Arg Type Checking/Test_TStreamAdd_Read_UDINT.TcPOU
FUNCTION_BLOCK Test_TStreamAdd_Read_UDINT EXTENDS T_UnitTestBase
VAR
    Stream  : T_Stream(StreamLength := 2);
    ArgType : E_ArgTypeId := E_ArgTypeId.Type_UDINT;
END_VAR

{attribute 'analysis' := '-33'} // inhibit unused variable warning
METHOD RunTest
IF Retest THEN
    SUPER^.Init();
END_IF

IF TestCompleted THEN
    RETURN;
END_IF

F_Inc(CycleCount);
IF CycleCount > 1000 THEN
    Fail(Message := 'Timeout');
END_IF

Stream.Init(2);

// add a UDINT...
Stream.SetNextArgTypeId(ArgType);
Stream.Add_UDINT(12345678);

Stream.SetReadPosition(0);

// check next arg type is correct...
AssertEquals_INT(Expected     := ArgType,
                           Actual       := Stream.GetNextArgTypeId(),
                           Message := 'Stream.GetNextArgTypeId()');

// check next value...	
AssertEquals_UDINT(Expected     := 12345678,
                             Actual       := Stream.Read_UDINT(),
                             Message := 'Stream.Read_UDINT()');

// check we are at the end of the stream..							
AssertEquals_UDINT(Expected     := Stream.StreamLength,
                             Actual       := Stream.ReadPosition,
                             Message := 'Stream.ReadPosition');

TestCompleted := TRUE;
END_METHOD

END_FUNCTION_BLOCK

// ---- Unit Tests/Stream/With Arg Type Checking/Test_TStreamAdd_Read_UINT.TcPOU
FUNCTION_BLOCK Test_TStreamAdd_Read_UINT EXTENDS T_UnitTestBase
VAR
    Stream  : T_Stream(StreamLength := 2);
    ArgType : E_ArgTypeId := E_ArgTypeId.Type_UINT;
END_VAR

{attribute 'analysis' := '-33'} // inhibit unused variable warning
METHOD RunTest
IF Retest THEN
    SUPER^.Init();
END_IF

IF TestCompleted THEN
    RETURN;
END_IF

F_Inc(CycleCount);
IF CycleCount > 1000 THEN
    Fail(Message := 'Timeout');
END_IF

Stream.Init(2);

// add a UINT...
Stream.SetNextArgTypeId(ArgType);
Stream.Add_UINT(4567);

Stream.SetReadPosition(0);

// check next arg type is correct...
AssertEquals_INT(Expected     := ArgType,
                           Actual       := Stream.GetNextArgTypeId(),
                           Message := 'Stream.GetNextArgTypeId()');

// check next value...	
AssertEquals_UINT(Expected     := 4567,
                            Actual       := Stream.Read_UINT(),
                            Message := 'Stream.Read_UINT()');

// check we are at the end of the stream..							
AssertEquals_UDINT(Expected     := Stream.StreamLength,
                             Actual       := Stream.ReadPosition,
                             Message := 'Stream.ReadPosition');

TestCompleted := TRUE;
END_METHOD

END_FUNCTION_BLOCK

// ---- Unit Tests/Stream/With Arg Type Checking/Test_TStreamAdd_Read_ULINT.TcPOU
FUNCTION_BLOCK Test_TStreamAdd_Read_ULINT EXTENDS T_UnitTestBase
VAR
    Stream  : T_Stream(StreamLength := 2);
    ArgType : E_ArgTypeId := E_ArgTypeId.Type_ULINT;
END_VAR

{attribute 'analysis' := '-33'} // inhibit unused variable warning
METHOD RunTest
IF Retest THEN
    SUPER^.Init();
END_IF

IF TestCompleted THEN
    RETURN;
END_IF

F_Inc(CycleCount);
IF CycleCount > 1000 THEN
    Fail(Message := 'Timeout');
END_IF


Stream.Init(2);

// add a ULINT...
Stream.SetNextArgTypeId(ArgType);
Stream.Add_ULINT(123456789);

Stream.SetReadPosition(0);

// check next arg type is correct...
AssertEquals_INT(Expected     := ArgType,
                           Actual       := Stream.GetNextArgTypeId(),
                           Message := 'Stream.GetNextArgTypeId()');

// check next value...	
AssertEquals_ULINT(Expected     := 123456789,
                             Actual       := Stream.Read_ULINT(),
                             Message := 'Stream.Read_ULINT()');

// check we are at the end of the stream..							
AssertEquals_UDINT(Expected     := Stream.StreamLength,
                             Actual       := Stream.ReadPosition,
                             Message := 'Stream.ReadPosition');

TestCompleted := TRUE;
END_METHOD

END_FUNCTION_BLOCK
